FUNCTION_BLOCK CompositeBlock
  FBS
    BaseBlock1 : BaseBlock;
    BaseBlock2 : BaseBlock;
    BaseBlock3 : BaseBlock;
    EA_2_router : EA_2_router;
    EA_network1_0 : EA_network1;
    EA_network1_1 : EA_network1;
    EA_network2_0 : EA_network2;
    EA_network2_1 : EA_network2;
  END_FBS
  ADAPTER_CONNECTIONS
    BaseBlock1.plug TO EA_2_router.socket;
    EA_2_router.plug_0 TO EA_network1_0.Socket_Connection;
    EA_2_router.plug_1 TO EA_network1_1.Socket_Connection;
    EA_network1_0.Plug_Connection TO EA_network2_0.Socket_Connection;
    EA_network2_0.Plug_Connection TO BaseBlock2.socket;
    EA_network1_1.Plug_Connection TO EA_network2_1.Socket_Connection;
    EA_network2_1.Plug_Connection TO BaseBlock3.socket;
  END_CONNECTIONS
END_FUNCTION_BLOCK
